% RSLogix 500 project CH6Q12.RSS, saved by version 8.30.00.16 %
PROJECT "CH6Q12"    % processor: Bul.1763 MicroLogix 1100 Series B %

PROGRAM FILES
  LAD 2   3 rungs

DATA FILES
  O0 OUTPUT  4 elements
  I1 INPUT  6 elements
  S2 STATUS  66 elements
  B3 BINARY  1 elements
  T4 TIMER  1 elements
  C5 COUNTER  1 elements
  R6 CONTROL  1 elements
  N7 INTEGER  1 elements
  F8 FLOAT  1 elements

LADDER 2
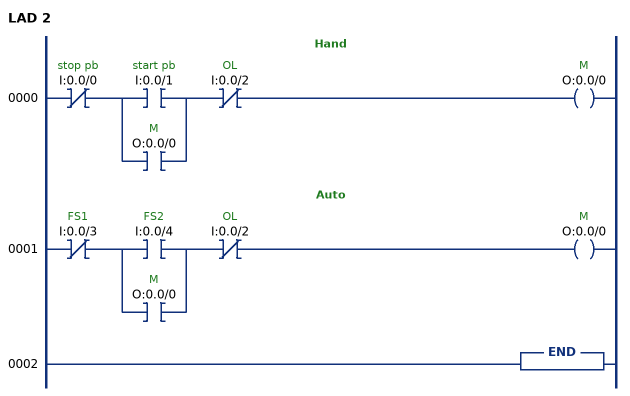
% Rung: 0 %
% TITLE: Hand %
SOR XIO I:0.0/0 BST XIC I:0.0/1 NXB XIC O:0.0/0 BND XIO I:0.0/2 OTE O:0.0/0 EOR
%   I:0.0/0  "stop pb" %
%   I:0.0/1  "start pb" %
%   O:0.0/0  "M" %
%   I:0.0/2  "OL" %
% Rung: 1 %
% TITLE: Auto %
SOR XIO I:0.0/3 BST XIC I:0.0/4 NXB XIC O:0.0/0 BND XIO I:0.0/2 OTE O:0.0/0 EOR
%   I:0.0/3  "FS1" %
%   I:0.0/4  "FS2" %
%   O:0.0/0  "M" %
%   I:0.0/2  "OL" %
% Rung: 2 %
SOR END EOR
